{attribute 'linkalways'}
{attribute 'no_explicit_call' := 'This FB is a CLASS and must be accessed using methods or properties'}
{attribute 'enable_dynamic_creation'}
FUNCTION_BLOCK _TcVnSize2_DINT EXTENDS StructuredDatatypeBase
VAR
    localData : TcVnSize2_DINT;
    activeData : REFERENCE TO TcVnSize2_DINT REF= localData;
    _nWidth : _DINT(localData.nWidth);
    _nHeight : _DINT(localData.nHeight);
END_VAR

PROPERTY PUBLIC Address : PVOID
GET
Address := ADR(activeData);
END_GET
END_PROPERTY

METHOD PUBLIC ClearReference
VAR_INPUT
END_VAR
activeData REF= localData;
SetMemberReference();
END_METHOD

METHOD PUBLIC Clone : I_Datatype
VAR
    pClone : POINTER TO _TcVnSize2_DINT;
END_VAR
pClone := __NEW(_TcVnSize2_DINT);
IF pClone = 0 THEN
    RETURN;
END_IF
pClone^.TryCopyFrom(THIS^);
Clone := pClone^;
END_METHOD

METHOD FB_init : BOOL
VAR_INPUT
	bInitRetains : BOOL; // if TRUE, the retain variables are initialized (warm start / cold start)
	bInCopyCode : BOOL;  // if TRUE, the instance afterwards gets moved into the copy code (online change)
END_VAR
SetMemberReference();
AddMember('nWidth', _nWidth);
AddMember('nHeight', _nHeight);
END_METHOD

PROPERTY PUBLIC Identifier : T_MAXSTRING
GET
Identifier := 'TcVnSize2_DINT';
END_GET
END_PROPERTY

METHOD PUBLIC MakeReferenceTo
VAR_INPUT
	ReferenceTarget : REFERENCE TO TcVnSize2_DINT;
END_VAR
activeData REF= ReferenceTarget;
SetMemberReference();
END_METHOD

METHOD PROTECTED SetMemberReference
VAR_INPUT
END_VAR
_nWidth.MakeReferenceTo(activeData.nWidth);
_nHeight.MakeReferenceTo(activeData.nHeight);
END_METHOD

PROPERTY PUBLIC Size : UDINT
GET
Size := SIZEOF(activeData);
END_GET
END_PROPERTY

METHOD TryMakeReferenceTo : BOOL
VAR_INPUT
	Target : I_Datatype;
END_VAR
VAR
	pTargetData : POINTER TO TcVnSize2_DINT;
END_VAR
IF NOT IsEquivalentTo(Target) THEN
	RETURN;
END_IF

pTargetData := Target.Address;
activeData REF= pTargetData^;
SetMemberReference();
TryMakeReferenceTo := TRUE;
END_METHOD

PROPERTY PUBLIC Value : REFERENCE TO TcVnSize2_DINT
GET
Value REF= activeData;
END_GET
END_PROPERTY

PROPERTY PUBLIC nWidth : REFERENCE TO _DINT
GET
nWidth REF= _nWidth;
END_GET
END_PROPERTY

PROPERTY PUBLIC nHeight : REFERENCE TO _DINT
GET
nHeight REF= _nHeight;
END_GET
END_PROPERTY

END_FUNCTION_BLOCK

(* stored: Version 1.1.0.1, ProductVersion 3.1.4024.13
   POU _TcVnSize2_DINT: Id {753d18d3-3e67-4ab6-a39b-a6952f96b44b}, SpecialFunc None
   Folder Core: Id {de957aa9-a424-4be6-9daf-f0b626e31574}
   Folder Customize: Id {d74bb207-0aaf-4f0b-b3b2-ef148240551b}
   Folder Constructor: Id {57539431-4780-458f-8130-8a36def2b7ae}
   Folder Protected: Id {162d6ff4-57f5-46bf-aa1d-62f746e20261}
   Property Address: Id {02be928b-57f4-4ee4-b72b-83abf1fc6920}
   Get Get: Id {439e234b-9cef-441d-b3a1-61c728b5eab5}
   Method ClearReference: Id {51ff12fc-2151-4af7-ba98-4dfae7a50564}
   Method Clone: Id {e0ae7a14-3d3c-48fd-92f1-63020046bd31}
   Method FB_init: Id {76743c39-03e6-4c91-acde-f568a4b72d7e}
   Property Identifier: Id {6dad0d71-b667-4655-a153-4ad0039cc2b9}
   Get Get: Id {858b34c5-7471-489b-b593-948d4536d45f}
   Method MakeReferenceTo: Id {ed57acd9-853a-46dc-a0c9-30deee5d72fa}
   Method SetMemberReference: Id {34379f6d-1eeb-4673-8027-152b4e6cbfc6}
   Property Size: Id {1b0bcc30-b542-4e11-987f-d8045a6bf665}
   Get Get: Id {e637d0ef-6c7e-4bea-aa0f-ab92d3082ccb}
   Method TryMakeReferenceTo: Id {0ba7aae6-04b7-4de5-b71f-b1c96d459dd2}
   Property Value: Id {0cd11b90-9f54-40f5-957a-8b5470f46108}
   Get Get: Id {2106594b-8c40-42b1-85d0-7be988ddbaf9}
   Property nWidth: Id {4201d214-a9bf-4f30-8258-627926fbc0d3}
   Get Get: Id {5f86a31b-3929-46da-b49e-0e3e77b416af}
   Property nHeight: Id {808e5b58-bc0f-472f-96ab-777f90c89146}
   Get Get: Id {58b1c480-31c7-4879-90e5-5c2f86a9b546} *)
